///#########################################################
///Function block to read and write axis parameters 
/// Library:
/// Tc2_MC2.lib
///
/// Global Variables:
///
/// Data types:
///
/// External functions:
///
///###########################################################
FUNCTION_BLOCK FB_ReadWriteParameter
VAR
	fbSet_RTRIG: R_TRIG;
	fbWriteParameter: MC_WriteParameter;
	fbReadParameter: MC_ReadParameter;
END_VAR
VAR_INPUT
	iParameterNumber: AxisParameters;
	fWriteParameter: LREAL;
	bSet: BOOL;
END_VAR
VAR_OUTPUT
	fReadParameter: LREAL;
END_VAR

VAR_IN_OUT
    stAxisStruct: ST_AxisStruct;
END_VAR


//Write Parameter
fbSet_RTRIG(clk := bSet);
fbWriteParameter( Axis := stAxisStruct.Axis, Execute := fbSet_RTRIG.Q, ParameterNumber := iParameterNumber, Value := fWriteParameter);

//Read Parameter
fbReadParameter( Axis := stAxisStruct.Axis, Enable := TRUE, ParameterNumber := iParameterNumber, ReadMode := 2);

IF NOT fbReadParameter.Error THEN
	fReadParameter := fbReadParameter.Value;
END_IF

END_FUNCTION_BLOCK

(* stored: Version 1.1.0.1, ProductVersion 3.1.4024.0
   POU FB_ReadWriteParameter: Id {c67413c7-a2ec-4895-814c-5b6c8c0c7aa9}, SpecialFunc None *)
